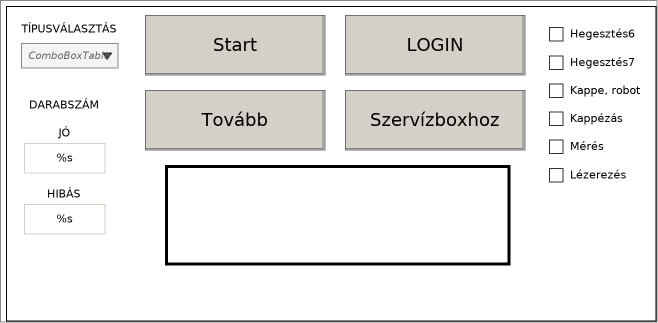
VISUALIZATION Termeles2  // 658x323
    Rectangle (6,6 650x315)
    Button (145,15 180x60), "Start"
        OnMouseUp: execute { AUTOMATA.iState2:=1; }
    Button (145,90 180x60), "Tovább"
        OnMouseUp: execute { AUTOMATA.bContinue2:=TRUE; }
    Button (345,90 180x60), "STOP"
        OnMouseUp: execute {
            AUTOMATA.bContinue2:=FALSE;
            AUTOMATA.iState2:=0;
            AUTOMATA.bWelderReservedBy2:=FALSE;
            AUTOMATA.bRobotReservedBy2:=FALSE;
        }
    Button (345,90 180x60), "Szervízboxhoz"
        OnMouseUp: execute { AUTOMATA.iState2:=100; }
    Textfield (24,143 81x30), "%s", text variable: GVL.nGoodProductCount, input disabled if: TRUE
    Label (52,118 25x30), "JÓ"
    Textfield (24,204 81x30), "%s", text variable: GVL.nBadProductCount, input disabled if: TRUE
    Label (43,179 42x30), "HIBÁS"
    Label (23,90 82x30), "DARABSZÁM"
    Label (14,14 110x30), "TÍPUSVÁLASZTÁS"
    Button (345,15 180x60), "LOGIN"
        OnMouseClick: VisuUserMgmt Type=Login
    RoundedRectangle (235,190 215x50), text list: 'ErrorList2', text index: AUTOMATA.iState2
    Group (547,19 105x171)
        Checkbox (0,141 105x30), "Lézerezés", variable: GVL.bJelolesBe, input disabled if: AUTOMATA.bFolyamatBeallitas2Tiltva
        Checkbox (0,0 105x30), "Hegesztés6", variable: GVL.bHegesztes6Be, input disabled if: AUTOMATA.bFolyamatBeallitas2Tiltva
        Checkbox (0,29 105x29), "Hegesztés7", variable: GVL.bHegesztes7Be, input disabled if: AUTOMATA.bFolyamatBeallitas2Tiltva
        Checkbox (0,57 105x29), "Kappe, robot", variable: GVL.bRobotKappeBe, input disabled if: AUTOMATA.bFolyamatBeallitas2Tiltva
        Checkbox (0,85 105x29), "Kappézás", variable: GVL.bKappeBe, input disabled if: AUTOMATA.bFolyamatBeallitas2Tiltva
        Checkbox (0,113 105x29), "Mérés", variable: GVL.bMeresBe, input disabled if: AUTOMATA.bFolyamatBeallitas2Tiltva
    Label (265,160 145x30), "JELENLEGI FOLYAMAT:"
    RoundedRectangle (165,165 345x100), text list: 'ErrorList1', text index: AUTOMATA.iState
    ComboBoxTable (21,43 97x25), variable: GVL.iSelectedProductType, data array: GVL.saProductTypes
        p3854506369: GVL.saProductTypes[INDEX]
END_VISUALIZATION

(* stored: Version 1.1.0.1, ProductVersion 3.1.4024.11
   Visu Termeles2: Id {4712a2ad-c94f-4993-a77e-78039cf45dd9} *)
